{attribute 'qualified_only'}
{attribute 'strict'}
{attribute 'to_string'}
TYPE E_ButtonColors :
(
	red,
	green,
	blue,
	white
);
END_TYPE

(* stored: Version 1.1.0.1, ProductVersion 3.1.4026.20
   DUT E_ButtonColors: Id {96595327-1893-4088-a0df-dc066d439257} *)
